# EPICS substitutions: gigeApp/Db/bld-hist.substitutions
#
# bld_hist.substitutions
#
# Uses the generated ai_hist_pattern.db template
# to create history waveforms for each of the
# specified PV's along with AVG, MAX, MIN,
# RMS, and StdDev for each history.
#
# Required Macros:
#	PV		 - PV name
# Optional Macros:
#	EGU		 - Engineering units, default to ""
#	RMS_LOLO - Low  alarm   limit for $(PV)_RMS, default 0
#	RMS_LOW  - Low  warning limit for $(PV)_RMS, default 0
#	RMS_HIGH - High warning limit for $(PV)_RMS, default 0
#	RMS_HIHI - High alarm   limit for $(PV)_RMS, default 0

# Example
file ai_hist_pattern.db
{
	pattern
	{	PV,										EGU		}
	{	"$(P)$(R)BLD1:AdjCtrMass_RBV",			"arb"	}
	{	"$(P)$(R)BLD1:AdjIntegral_RBV",			"arb"	}
	{	"$(P)$(R)BLD1:ArrayRate_RBV",			"Hz"	}
	{	"$(P)$(R)BLD1:HorizRawCtrMass_RBV",		"arb"	}
	{	"$(P)$(R)BLD1:HorizRawIntegral_RBV",	"arb"	}
}
